INTERFACE ITF_GroupElement_HMI

END_INTERFACE

(* stored: Version 1.1.0.1, ProductVersion 3.1.4024.15
   Itf ITF_GroupElement_HMI: Id {56ded6a8-c57d-4918-9207-29ee5c9f0bfe} *)
